PROGRAM P_BlockPad
VAR_INPUT
	NappiNumero: INT;
END_VAR
VAR
	Numero: INT;
	nRes: INT;
	n1: INT;
	n2: INT;
	n3: INT;
	
	eNappi : E_NappienNumerointi;
	(*
	r2 : E_Nappinumerot.Vipu1;
	r3 : E_Nappinumerot.Vipu2; *)
	
	Numero2: INT;
	fbBlock: FB_ButtonBox;
	FB_Block_0: FB_ButtonBox;
	fbBlock_0: FB_ButtonBox;
	NappiOhje: INT;
END_VAR


//F_Sample(nVar1:=1,nVar2:=44,nVar3:=3);
Numero := F_Sample(1,1,44);
P_BlockPad(NappiNumero:= Numero);

P_BlockPad(NappiNumero := NappiOhje);



Numero := NappiNumero;
n1 := 44; 
n2 := 4;
n3 := 83;
nRes := F_Sample(n1,n2,n3);
eNappi := E_NappienNumerointi.Vipu2;
// Numero2 := r1 + r2 + r3;
(*
fbBlock(
iInput1:= IO.BOX_IN[1] ,
iInput2:= IO.BOX_IN[2], 
iInput3:= IO.BOX_IN[3], 
oLight1=> IO.BOX_OUT[1]
);

*)

(*
IF IO.BOX_IN[1] THEN
 Numero := Numero +1;
 IO.BOX_OUT[1] := TRUE;
END_IF
*)

END_PROGRAM

(* stored: Version 1.1.0.1, ProductVersion 3.1.4024.10
   POU P_BlockPad: Id {8a1efacf-3fcd-461c-b49b-df5e51cc6e16}, SpecialFunc None *)
